PopupScreen "Option3" 400x400
   Rectangle "Rectangle_6" at 54,54 size 27x7
      Appearance <- "Data_7SEG_DIV"
   Rectangle "Rectangle_7" at 80,60 size 8x34
      Appearance <- "Data_7SEG_DIV"
   Rectangle "Rectangle_8" at 54,93 size 27x7
      Appearance <- "Data_7SEG_DIV"
   Rectangle "Rectangle_9" at 81,99 size 8x30
      Appearance <- "Data_7SEG_DIV"
   Rectangle "Rectangle_10" at 53,128 size 29x8
      Appearance <- "Data_7SEG_DIV"
   Rectangle "Rectangle_11" at 47,99 size 8x30
      Appearance <- "Data_7SEG_DIV"
   Rectangle "Rectangle_12" at 46,60 size 8x33
      Appearance <- "Data_7SEG_DIV"
   Rectangle "Rectangle_13" at 102,55 size 26x8
      Appearance <- "Data_7SEG_MOD"
   Rectangle "Rectangle_14" at 127,62 size 8x32
      Appearance <- "Data_7SEG_MOD"
   Rectangle "Rectangle_16" at 102,93 size 26x7
      Appearance <- "Data_7SEG_MOD"
   Rectangle "Rectangle_17" at 128,100 size 8x29
      Appearance <- "Data_7SEG_MOD"
   Rectangle "Rectangle_18" at 102,128 size 27x8
      Appearance <- "Data_7SEG_MOD"
   Rectangle "Rectangle_19" at 95,98 size 8x31
      Appearance <- "Data_7SEG_MOD"
   Rectangle "Rectangle_20" at 95,62 size 8x32
      Appearance <- "Data_7SEG_MOD"
   Rectangle "Rectangle_22" at 185,57 size 26x7
      Appearance <- "Data_7SEG_DIV_B"
   Rectangle "Rectangle_23" at 210,63 size 8x30
      Appearance <- "Data_7SEG_DIV_B"
   Rectangle "Rectangle_24" at 185,92 size 26x7
      Appearance <- "Data_7SEG_DIV_B"
   Rectangle "Rectangle_25" at 210,98 size 8x29
      Appearance <- "Data_7SEG_DIV_B"
   Rectangle "Rectangle_26" at 186,126 size 25x7
      Appearance <- "Data_7SEG_DIV_B"
   Rectangle "Rectangle_27" at 178,99 size 8x28
      Appearance <- "Data_7SEG_DIV_B"
   Rectangle "Rectangle_28" at 178,63 size 8x30
      Appearance <- "Data_7SEG_DIV_B"
   Rectangle "Rectangle_29" at 239,57 size 26x7
      Appearance <- "Data_7SEG_MOD_B"
   Rectangle "Rectangle_30" at 264,63 size 8x30
      Appearance <- "Data_7SEG_MOD_B"
   Rectangle "Rectangle_31" at 239,92 size 27x7
      Appearance <- "Data_7SEG_MOD_B"
   Rectangle "Rectangle_32" at 265,98 size 8x28
      Appearance <- "Data_7SEG_MOD_B"
   Rectangle "Rectangle_33" at 239,125 size 27x8
      Appearance <- "Data_7SEG_MOD_B"
   Rectangle "Rectangle_34" at 232,98 size 8x28
      Appearance <- "Data_7SEG_MOD_B"
   Rectangle "Rectangle_35" at 232,63 size 8x30
      Appearance <- "Data_7SEG_MOD_B"
   TextField "Text field_11" at 54,141 size 63x29; Text 'Side A'
   TextField "Text field_12" at 197,141 size 64x30; Text 'Side B'
*)

(* ===== HMI "HMI_RT_3" =====
system functions are stored by id; their names below are inferred from use
connection "HMI_Connection_8": S71200_TCP_IP, SCADA_S7_1500_OMS

screen "Screen_1" 1024x600
   GraphicView "Graphic view_2" at 949,4 size 70x69; Picture "Close_Button"
      on Click: "OnClick"
   Clock "Clock_1" at 780,7 size 178x25
*)